// TIA Portal V16 export
// export: Created 2021-04-13T11:10:15.3878321Z, ExportSetting WithDefaults, DisplayName Totally Integrated Automation Portal, DisplayVersion V16, DisplayName TIA Portal Version Control Interface, DisplayVersion V16, DisplayName TIA Portal Openness, DisplayVersion V16, DisplayName STEP 7 Professional, DisplayVersion V16, DisplayName STEP 7 Safety, DisplayVersion V16, DisplayName WinCC Unified SCADA Engineering System, DisplayVersion V16
FUNCTION_BLOCK "weightModule_AM"   // FB12, LAD
{ S7_Optimized_Access := 'TRUE' }
VERSION : 0.1
// stored: AutoNumber true, IsIECCheckEnabled false, IsRetainMemResEnabled false, MemoryReserve 100, SetENOAutomatically false, UDAEnableTagReadback false
   VAR_IN_OUT
      currentWeight : Array[0..12] of Real;   // текущий вес
      stableWeight : Array[0..12] of "stableWeight";   // массивы стабильных весов
   END_VAR
   VAR
      tonSetStableWeight : Array[0..12] of TON_TIME;   // выдержка для переноса текущего веса в разряд стабильных
      prevWeight : Array[0..12] of Real;   // предыдущий вес
      runTaimerStableWeight : Array[0..12] of Bool;
      RS_TRIG_openBunker : Array[0..12] of Bool;   // триггер что бункера были открыты
   END_VAR
   VAR_TEMP
      i : DInt;
   END_VAR
BEGIN

REGION Network 1 (SCL)
   #i := 0;
   FOR #i := 1 TO 12 DO

       IF "hmi".weightLine[#i].stateLeftValveWeightPocket OR "hmi".weightLine[#i].stateRightValveWeightPocket THEN
           #RS_TRIG_openBunker[#i] := true;//фиксируем что произошло открытие бункеров
       END_IF;
       IF NOT("hmi".weightLine[#i].stateLeftValveWeightPocket) AND NOT("hmi".weightLine[#i].stateRightValveWeightPocket) THEN
           #RS_TRIG_openBunker[#i] := false;//если бункера закрыты, то сбрасываем фиксацию о их открытии
       END_IF;

       IF NOT (#RS_TRIG_openBunker[#i]) THEN

           IF (#prevWeight[#i] - 10) <= #currentWeight[#i] AND #currentWeight[#i] <= (#prevWeight[#i] + 10) THEN
               #runTaimerStableWeight[#i] := true;
           ELSE
               #runTaimerStableWeight[#i] := false;
               #prevWeight[#i] := #currentWeight[#i];
           END_IF;
           #tonSetStableWeight[#i](IN := #runTaimerStableWeight[#i],
                                   PT := t#20ms);

       ELSE
           #currentWeight[#i] := 0;
           #prevWeight[#i]:= 0;
       END_IF;

       IF #tonSetStableWeight[#i].Q OR #RS_TRIG_openBunker[#i] THEN
           IF #currentWeight[#i] <> "signalKVSStation".stableWeight[#i].weight[0] THEN
               "pushToArray"(addValue := #currentWeight[#i],
                             "array" := #stableWeight[#i].weight);
           END_IF;
           #runTaimerStableWeight[#i] := false;
       END_IF;


   END_FOR;
END_REGION
END_FUNCTION_BLOCK
